// TIA Portal V20 export
// export: Created 2025-12-01T14:57:20.3173297Z, ExportSetting None, DisplayName Totally Integrated Automation Portal, DisplayVersion V20 Update 3, DisplayName TIA Portal Openness, DisplayVersion V20 Update 3, DisplayName TIA Portal Version Control Interface, DisplayVersion V20 Update 3, DisplayName STEP 7 Professional, DisplayVersion V20 Update 3, DisplayName STEP 7 Safety, DisplayVersion V20 Update 2, DisplayName WinCC Basic/Comfort/Advanced, DisplayVersion V20 Update 3, DisplayName WinCC Professional, DisplayVersion V20 Update 3, DisplayName WinCC Unified, DisplayVersion V20 Update 3
DATA_BLOCK "DB870_ConversorEventos"   // DB870
{ S7_Optimized_Access := 'FALSE' }
// stored: AutoNumber false
   VAR
      Etiqueta_A_Valor : Array[1.."CTE_MaxArrayConversion"] of Struct
         Etiqueta : DWord;
         Valor : Int;
      END_STRUCT;
      Valor_A_Etiqueta : Array[1.."CTE_MaxArrayConversion"] of Struct
         Valor : Int;
         Etiqueta : DWord;
      END_STRUCT;
      EventosRecibidos : Array[1.."CTE_MaxArrayConversion"] of DWord;
      AtributosRecibidosDeUTs : Array[1.."CTE_MaxArrayConversion"] of DWord;
      AtributosRecibidosDeDispositivos : Array[1.."CTE_MaxArrayConversion"] of DWord;
      AtributosRecibidosDeRouter : Array[1.."CTE_MaxArrayConversion"] of DWord;
      AtributosRecibidosDeQuimarox : Array[1.."CTE_MaxArrayConversion"] of DWord;
      AtributosRecibidosDeReset : Array[1.."CTE_MaxArrayConversion"] of DWord;
   END_VAR
BEGIN
   Etiqueta_A_Valor[1].Etiqueta := 'MARC';
   Etiqueta_A_Valor[2].Etiqueta := 'PARO';
   Etiqueta_A_Valor[3].Etiqueta := 'REAR';
   Etiqueta_A_Valor[4].Etiqueta := 'RESE';
   Etiqueta_A_Valor[5].Etiqueta := 'BLAN';
   Etiqueta_A_Valor[6].Etiqueta := 'AUTO';
   Etiqueta_A_Valor[7].Etiqueta := 'MANU';
   Etiqueta_A_Valor[8].Etiqueta := 'ERRO';
   Etiqueta_A_Valor[9].Etiqueta := 'CCPI';
   Etiqueta_A_Valor[10].Etiqueta := 'CBOX';
   Etiqueta_A_Valor[11].Etiqueta := 'MESA';
   Etiqueta_A_Valor[12].Etiqueta := 'MAQU';
   Etiqueta_A_Valor[13].Etiqueta := 'EURO';
   Etiqueta_A_Valor[14].Etiqueta := 'MEDI';
   Etiqueta_A_Valor[15].Etiqueta := 'CUAR';
   Etiqueta_A_Valor[16].Etiqueta := 'CHEE';
   Etiqueta_A_Valor[17].Etiqueta := 'PARM';
   Etiqueta_A_Valor[18].Etiqueta := '2CUA';
   Etiqueta_A_Valor[19].Etiqueta := 'AMER';
   Etiqueta_A_Valor[20].Etiqueta := 'LPR_';
   Etiqueta_A_Valor[21].Etiqueta := 'CA_1';
   Etiqueta_A_Valor[22].Etiqueta := 'CA_2';
   Etiqueta_A_Valor[23].Etiqueta := '_SI_';
   Etiqueta_A_Valor[24].Etiqueta := '_NO_';
   Etiqueta_A_Valor[25].Etiqueta := 'BALI';
   Etiqueta_A_Valor[26].Etiqueta := 'LLAV';
   Etiqueta_A_Valor[27].Etiqueta := 'SETA';
   Etiqueta_A_Valor[28].Etiqueta := 'BARR';
   Etiqueta_A_Valor[29].Etiqueta := 'PUER';
   Etiqueta_A_Valor[30].Etiqueta := 'LINP';
   Etiqueta_A_Valor[31].Etiqueta := 'MADE';
   Etiqueta_A_Valor[32].Etiqueta := 'ROJO';
   Etiqueta_A_Valor[33].Etiqueta := 'AZUL';
   Etiqueta_A_Valor[34].Etiqueta := 'VERD';
   Etiqueta_A_Valor[35].Etiqueta := 'ERRR';
   Etiqueta_A_Valor[36].Etiqueta := 'NENC';
   Etiqueta_A_Valor[37].Etiqueta := 'INIC';
   Etiqueta_A_Valor[38].Etiqueta := 'STAT';
   Etiqueta_A_Valor[39].Etiqueta := 'POSI';
   Etiqueta_A_Valor[40].Etiqueta := 'VTDC';
   Etiqueta_A_Valor[41..42].Etiqueta := 'ELEV';
   Etiqueta_A_Valor[43].Etiqueta := 'REMO';
   Etiqueta_A_Valor[44].Etiqueta := 'APIL';
   Etiqueta_A_Valor[45].Etiqueta := 'VTDC';
   Etiqueta_A_Valor[46].Etiqueta := 'ENFA';
   Etiqueta_A_Valor[47].Etiqueta := 'ETIQ';
   Etiqueta_A_Valor[48].Etiqueta := 'FLEJ';
   Etiqueta_A_Valor[1].Valor := 6;
   Etiqueta_A_Valor[2].Valor := 5;
   Etiqueta_A_Valor[3].Valor := 2;
   Etiqueta_A_Valor[4].Valor := 4;
   Etiqueta_A_Valor[5].Valor := 3;
   Etiqueta_A_Valor[6].Valor := 8;
   Etiqueta_A_Valor[7].Valor := 9;
   Etiqueta_A_Valor[8].Valor := 1;
   Etiqueta_A_Valor[9].Valor := 50;
   Etiqueta_A_Valor[10].Valor := 40;
   Etiqueta_A_Valor[11].Valor := 60;
   Etiqueta_A_Valor[12].Valor := 70;
   Etiqueta_A_Valor[13].Valor := 1;
   Etiqueta_A_Valor[14].Valor := 2;
   Etiqueta_A_Valor[15].Valor := 3;
   Etiqueta_A_Valor[16].Valor := 4;
   Etiqueta_A_Valor[17].Valor := 5;
   Etiqueta_A_Valor[18].Valor := 6;
   Etiqueta_A_Valor[19].Valor := 7;
   Etiqueta_A_Valor[20].Valor := 8;
   Etiqueta_A_Valor[21].Valor := 100;
   Etiqueta_A_Valor[22].Valor := 110;
   Etiqueta_A_Valor[23].Valor := 2001;
   Etiqueta_A_Valor[24].Valor := 2002;
   Etiqueta_A_Valor[25].Valor := 1000;
   Etiqueta_A_Valor[26].Valor := 1001;
   Etiqueta_A_Valor[27].Valor := 1002;
   Etiqueta_A_Valor[28].Valor := 1003;
   Etiqueta_A_Valor[29].Valor := 1004;
   Etiqueta_A_Valor[30].Valor := 1005;
   Etiqueta_A_Valor[31].Valor := 1;
   Etiqueta_A_Valor[32].Valor := 2;
   Etiqueta_A_Valor[33].Valor := 3;
   Etiqueta_A_Valor[34].Valor := 4;
   Etiqueta_A_Valor[35].Valor := 7000;
   Etiqueta_A_Valor[36].Valor := 7001;
   Etiqueta_A_Valor[37].Valor := 7002;
   Etiqueta_A_Valor[38].Valor := 5000;
   Etiqueta_A_Valor[39].Valor := 5001;
   Etiqueta_A_Valor[40].Valor := 74;
   Etiqueta_A_Valor[41..42].Valor := 71;
   Etiqueta_A_Valor[43].Valor := 72;
   Etiqueta_A_Valor[44].Valor := 73;
   Etiqueta_A_Valor[45].Valor := 74;
   Etiqueta_A_Valor[46].Valor := 75;
   Etiqueta_A_Valor[47].Valor := 76;
   Etiqueta_A_Valor[48].Valor := 77;
   Valor_A_Etiqueta[1].Valor := 1;
   Valor_A_Etiqueta[2].Valor := 2;
   Valor_A_Etiqueta[3].Valor := 4;
   Valor_A_Etiqueta[4].Valor := 5;
   Valor_A_Etiqueta[5].Valor := 6;
   Valor_A_Etiqueta[6].Valor := 11;
   Valor_A_Etiqueta[7].Valor := 12;
   Valor_A_Etiqueta[8].Valor := 14;
   Valor_A_Etiqueta[9].Valor := 50;
   Valor_A_Etiqueta[10].Valor := 40;
   Valor_A_Etiqueta[11].Valor := 60;
   Valor_A_Etiqueta[12].Valor := 70;
   Valor_A_Etiqueta[13].Valor := 21;
   Valor_A_Etiqueta[14].Valor := 22;
   Valor_A_Etiqueta[15].Valor := 121;
   Valor_A_Etiqueta[16].Valor := 122;
   Valor_A_Etiqueta[17].Valor := 123;
   Valor_A_Etiqueta[18].Valor := 124;
   Valor_A_Etiqueta[19].Valor := 125;
   Valor_A_Etiqueta[20].Valor := 1000;
   Valor_A_Etiqueta[21].Valor := 1001;
   Valor_A_Etiqueta[22].Valor := 1002;
   Valor_A_Etiqueta[23].Valor := 1011;
   Valor_A_Etiqueta[24].Valor := 1012;
   Valor_A_Etiqueta[25].Valor := 1013;
   Valor_A_Etiqueta[26].Valor := 2001;
   Valor_A_Etiqueta[27].Valor := 2002;
   Valor_A_Etiqueta[28].Valor := 3001;
   Valor_A_Etiqueta[29].Valor := 3002;
   Valor_A_Etiqueta[30].Valor := 3003;
   Valor_A_Etiqueta[31].Valor := 3004;
   Valor_A_Etiqueta[32].Valor := 3005;
   Valor_A_Etiqueta[33].Valor := 3006;
   Valor_A_Etiqueta[34].Valor := 3007;
   Valor_A_Etiqueta[35].Valor := 3008;
   Valor_A_Etiqueta[36].Valor := 3010;
   Valor_A_Etiqueta[37].Valor := 3011;
   Valor_A_Etiqueta[38].Valor := 3101;
   Valor_A_Etiqueta[39].Valor := 3102;
   Valor_A_Etiqueta[40].Valor := 3103;
   Valor_A_Etiqueta[41].Valor := 3104;
   Valor_A_Etiqueta[42].Valor := 71;
   Valor_A_Etiqueta[43].Valor := 72;
   Valor_A_Etiqueta[44].Valor := 73;
   Valor_A_Etiqueta[45].Valor := 74;
   Valor_A_Etiqueta[46].Valor := 75;
   Valor_A_Etiqueta[47].Valor := 76;
   Valor_A_Etiqueta[48].Valor := 77;
   Valor_A_Etiqueta[49].Valor := 126;
   Valor_A_Etiqueta[1].Etiqueta := 'MARC';
   Valor_A_Etiqueta[2].Etiqueta := 'PARO';
   Valor_A_Etiqueta[3..5].Etiqueta := 'ERRO';
   Valor_A_Etiqueta[6].Etiqueta := 'AUTO';
   Valor_A_Etiqueta[7].Etiqueta := 'MANT';
   Valor_A_Etiqueta[8].Etiqueta := 'MANU';
   Valor_A_Etiqueta[9].Etiqueta := 'CCPI';
   Valor_A_Etiqueta[10].Etiqueta := 'CBOX';
   Valor_A_Etiqueta[11].Etiqueta := 'MESA';
   Valor_A_Etiqueta[12].Etiqueta := 'MAQU';
   Valor_A_Etiqueta[13].Etiqueta := 'RESE';
   Valor_A_Etiqueta[14].Etiqueta := 'BLAN';
   Valor_A_Etiqueta[15].Etiqueta := 'RESE';
   Valor_A_Etiqueta[16].Etiqueta := 'BLOQ';
   Valor_A_Etiqueta[17].Etiqueta := 'RUTA';
   Valor_A_Etiqueta[18].Etiqueta := 'NDES';
   Valor_A_Etiqueta[19].Etiqueta := 'FUER';
   Valor_A_Etiqueta[20].Etiqueta := 'VACI';
   Valor_A_Etiqueta[21].Etiqueta := 'SEMI';
   Valor_A_Etiqueta[22].Etiqueta := 'LLEN';
   Valor_A_Etiqueta[23].Etiqueta := '_INI';
   Valor_A_Etiqueta[24].Etiqueta := '_FIN';
   Valor_A_Etiqueta[25].Etiqueta := 'ERRO';
   Valor_A_Etiqueta[26].Etiqueta := '__SI';
   Valor_A_Etiqueta[27].Etiqueta := '__NO';
   Valor_A_Etiqueta[28].Etiqueta := 'EURO';
   Valor_A_Etiqueta[29].Etiqueta := 'MEDI';
   Valor_A_Etiqueta[30].Etiqueta := 'CUAR';
   Valor_A_Etiqueta[31].Etiqueta := 'CHEE';
   Valor_A_Etiqueta[32].Etiqueta := 'PARM';
   Valor_A_Etiqueta[33].Etiqueta := '2CUA';
   Valor_A_Etiqueta[34].Etiqueta := 'AMER';
   Valor_A_Etiqueta[35].Etiqueta := 'LPR_';
   Valor_A_Etiqueta[36].Etiqueta := 'CA_1';
   Valor_A_Etiqueta[37].Etiqueta := 'CA_2';
   Valor_A_Etiqueta[38].Etiqueta := 'MADE';
   Valor_A_Etiqueta[39].Etiqueta := 'ROJO';
   Valor_A_Etiqueta[40].Etiqueta := 'AZUL';
   Valor_A_Etiqueta[41].Etiqueta := 'VERD';
   Valor_A_Etiqueta[42].Etiqueta := 'ELEV';
   Valor_A_Etiqueta[43].Etiqueta := 'REMO';
   Valor_A_Etiqueta[44].Etiqueta := 'APIL';
   Valor_A_Etiqueta[45].Etiqueta := 'VTDC';
   Valor_A_Etiqueta[46].Etiqueta := 'ENFA';
   Valor_A_Etiqueta[47].Etiqueta := 'ETIQ';
   Valor_A_Etiqueta[48].Etiqueta := 'FLEJ';
   Valor_A_Etiqueta[49].Etiqueta := 'ROBO';
   EventosRecibidos[1] := 'CREA';
   EventosRecibidos[2] := 'RUTA';
   EventosRecibidos[3] := 'DRUT';
   EventosRecibidos[4] := 'RETI';
   EventosRecibidos[5] := 'BORR';
   EventosRecibidos[6] := 'DATA';
   EventosRecibidos[7] := '?UT?';
   EventosRecibidos[8] := 'MOVE';
   EventosRecibidos[9] := 'DEMB';
   EventosRecibidos[10] := 'CSTA';
   EventosRecibidos[11] := 'DIDO';
   EventosRecibidos[12] := 'ORDE';
   EventosRecibidos[13] := 'BOET';
   EventosRecibidos[14] := 'BOBD';
   EventosRecibidos[15] := 'RUET';
   EventosRecibidos[16] := 'RUES';
   EventosRecibidos[17] := 'INIR';
   EventosRecibidos[18] := '?ST?';
   EventosRecibidos[19] := 'QCRE';
   EventosRecibidos[20] := 'QPR?';
   EventosRecibidos[21] := 'CHEQ';
   AtributosRecibidosDeUTs[1] := 'MCKY';
   AtributosRecibidosDeUTs[2] := 'MESA';
   AtributosRecibidosDeUTs[3] := 'RUTA';
   AtributosRecibidosDeUTs[4] := 'SALI';
   AtributosRecibidosDeUTs[5] := 'SSCC';
   AtributosRecibidosDeUTs[6] := 'GRUP';
   AtributosRecibidosDeUTs[7] := 'GCNT';
   AtributosRecibidosDeUTs[8] := 'GORD';
   AtributosRecibidosDeUTs[9] := 'FLEJ';
   AtributosRecibidosDeUTs[10] := 'ENFA';
   AtributosRecibidosDeUTs[11] := 'ETIQ';
   AtributosRecibidosDeUTs[12] := 'AMAR';
   AtributosRecibidosDeUTs[13] := 'PRES';
   AtributosRecibidosDeUTs[14] := 'NBUL';
   AtributosRecibidosDeUTs[15] := 'NTBU';
   AtributosRecibidosDeUTs[16] := 'PID_';
   AtributosRecibidosDeUTs[17] := 'TIPO';
   AtributosRecibidosDeUTs[18] := 'REMO';
   AtributosRecibidosDeUTs[19] := 'PILA';
   AtributosRecibidosDeUTs[20] := 'VACI';
   AtributosRecibidosDeUTs[21] := 'COTA';
   AtributosRecibidosDeUTs[22] := 'COTW';
   AtributosRecibidosDeUTs[23] := 'COTL';
   AtributosRecibidosDeUTs[24] := 'PESO';
   AtributosRecibidosDeUTs[25] := 'ALTO';
   AtributosRecibidosDeUTs[26] := 'ANCH';
   AtributosRecibidosDeUTs[27] := 'PROF';
   AtributosRecibidosDeUTs[28] := 'TACO';
   AtributosRecibidosDeUTs[29] := 'HUEC';
   AtributosRecibidosDeUTs[30] := 'HUER';
   AtributosRecibidosDeUTs[31] := 'COLO';
   AtributosRecibidosDeUTs[32] := 'PATI';
   AtributosRecibidosDeUTs[33] := 'LETI';
   AtributosRecibidosDeUTs[34] := 'SGAP';
   AtributosRecibidosDeUTs[35] := 'SGAE';
   AtributosRecibidosDeUTs[36] := 'SGAD';
   AtributosRecibidosDeUTs[37] := 'SGA_';
   AtributosRecibidosDeUTs[38] := 'RSLT';
   AtributosRecibidosDeUTs[39] := 'PDST';
   AtributosRecibidosDeUTs[40] := 'DEST';
   AtributosRecibidosDeUTs[41] := 'PALE';
   AtributosRecibidosDeDispositivos[1] := 'TIPO';
   AtributosRecibidosDeDispositivos[2] := 'NUME';
   AtributosRecibidosDeDispositivos[3] := 'NUES';
   AtributosRecibidosDeDispositivos[4] := 'HABI';
   AtributosRecibidosDeDispositivos[5] := 'PRIO';
   AtributosRecibidosDeDispositivos[6] := 'SONO';
   AtributosRecibidosDeDispositivos[7] := 'VERD';
   AtributosRecibidosDeDispositivos[8] := 'ROJO';
   AtributosRecibidosDeDispositivos[9] := 'AMAR';
   AtributosRecibidosDeDispositivos[10] := 'AZUL';
   AtributosRecibidosDeDispositivos[11] := 'MOTI';
   AtributosRecibidosDeDispositivos[12] := 'OPER';
   AtributosRecibidosDeDispositivos[13] := 'TEXT';
   AtributosRecibidosDeDispositivos[14] := 'HORQ';
   AtributosRecibidosDeDispositivos[15] := 'POSI';
   AtributosRecibidosDeRouter[1] := 'MESA';
   AtributosRecibidosDeRouter[2] := 'SSCC';
   AtributosRecibidosDeRouter[3] := 'SALI';
   AtributosRecibidosDeRouter[4] := 'DEST';
   AtributosRecibidosDeRouter[5] := 'NUME';
   AtributosRecibidosDeRouter[6] := 'HABI';
   AtributosRecibidosDeRouter[7] := 'ETES';
   AtributosRecibidosDeQuimarox[1] := 'MESA';
   AtributosRecibidosDeQuimarox[2] := 'PEIN';
   AtributosRecibidosDeQuimarox[3] := 'MCKY';
   AtributosRecibidosDeQuimarox[4] := 'ORIG';
   AtributosRecibidosDeQuimarox[5] := 'DEST';
   AtributosRecibidosDeQuimarox[6] := 'SSCC';
   AtributosRecibidosDeReset[1] := 'TIPO';
   AtributosRecibidosDeReset[2] := 'NUME';
   AtributosRecibidosDeReset[3] := 'OPER';
END_DATA_BLOCK
